INTERFACE I_AsynchronousRpcHandler EXTENDS __SYSTEM.IQueryInterface

METHOD Handle
VAR_INPUT
	Parameters : I_Deserializer;
	Response : I_AsynchronousRpcResponse;
END_VAR
END_METHOD

END_INTERFACE

(* stored: Version 1.1.0.1, ProductVersion 3.1.4026.13
   Itf I_AsynchronousRpcHandler: Id {f1cfa2fd-5bd3-0670-0bfe-bc15b5e54bd5}
   Method Handle: Id {a513e316-4e55-0699-139d-a1a2e557696a} *)
